TYPE Struct_OUT :
STRUCT
	bHeat1	:	BOOL;
	bOK		:	BOOL;
	
END_STRUCT
END_TYPE

(* stored: Version 1.1.0.1, ProductVersion 3.1.4024.16
   DUT Struct_OUT: Id {707ef7fd-c1ae-4985-aa0d-5254b2236ee0} *)
